(*
Implements the procedure for safely transitioning between device states by asserting the correct beam parameters for 
the state *)
FUNCTION_BLOCK BeamParameterTransitionManager
VAR_IN_OUT
	
	fbArbiter	:	FB_Arbiter;
	
END_VAR
VAR_INPUT
	i_TransitionAssertionID	:	UDINT := 0;
	i_stTransitionAssertion : ST_BeamParams := PMPS_GVL_BeamParams.cstSafeBeam; //Assertion required during transition (always safer than anything inbetween)
	
	i_nRequestedAssertionID	:	UDINT := 0;
	i_stRequestedAssertion	:	ST_BeamParams := PMPS_GVL_BeamParams.cstSafeBeam; //Requested assertion, change whenever
	
	i_xMoving	:	BOOL := FALSE; //Provide rising edge when device begins moving
	i_xDoneMoving	:	BOOL := FALSE; //Provide rising edge when device is done with a move
	
END_VAR
VAR_OUTPUT

	q_xTransitionAuthorized	:	BOOL := FALSE; //Rising edge indicating the device is safe to move, use as input to move execute (which requires a rising edge)

END_VAR

VAR
	nTargetAssertionID	:	UDINT := 0;
	stTargetAssertion	:	ST_BeamParams; //Current target assertion
	nCurrentAssertionID	:	UDINT := 0;
	
	xNewBP	:	BOOL;
	xTranBP	:	BOOL;
	xFinalBP	:	BOOL;
	
END_VAR

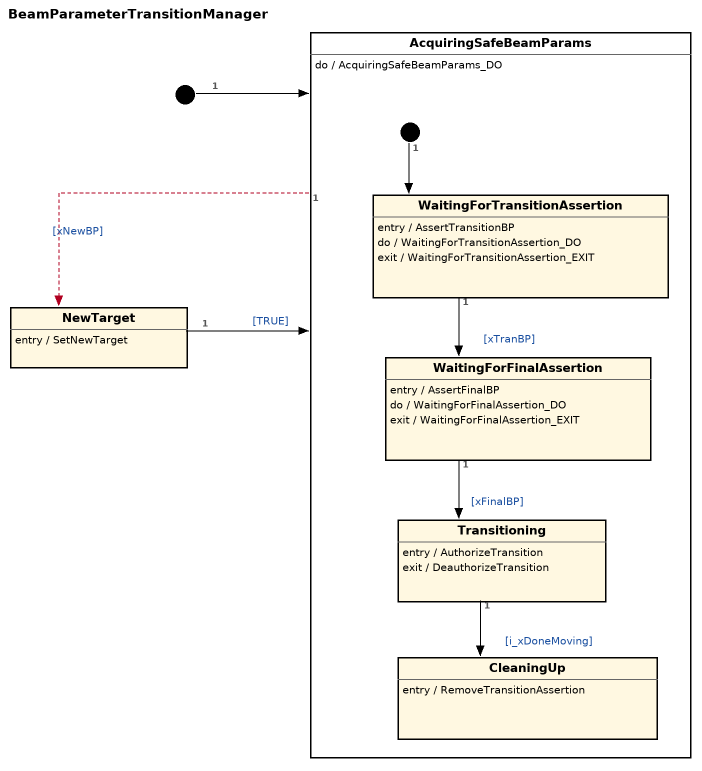
STATECHART BeamParameterTransitionManager  // abortable
    START StartState1_copy
    COMPOSITE STATE AcquiringSafeBeamParams
        do / AcquiringSafeBeamParams_DO
        START StartState1
        STATE WaitingForTransitionAssertion
            entry / AssertTransitionBP
            do / WaitingForTransitionAssertion_DO
            exit / WaitingForTransitionAssertion_EXIT
        STATE WaitingForFinalAssertion
            entry / AssertFinalBP
            do / WaitingForFinalAssertion_DO
            exit / WaitingForFinalAssertion_EXIT
        STATE Transitioning
            entry / AuthorizeTransition
            exit / DeauthorizeTransition
        STATE CleaningUp
            entry / RemoveTransitionAssertion
        StartState1 -> WaitingForTransitionAssertion  // priority 1, on completion
        WaitingForTransitionAssertion -> WaitingForFinalAssertion [xTranBP] // priority 1, rising edge
        WaitingForFinalAssertion -> Transitioning [xFinalBP] // priority 1, rising edge
        Transitioning -> CleaningUp [i_xDoneMoving] // priority 1, rising edge
    END_STATE
    STATE NewTarget
        entry / SetNewTarget
    StartState1_copy -> AcquiringSafeBeamParams  // priority 1, on completion
    AcquiringSafeBeamParams -> NewTarget [xNewBP] // priority 1, exception, rising edge
    NewTarget -> AcquiringSafeBeamParams [TRUE] // priority 1
END_STATECHART

ACTION AcquiringSafeBeamParams_DO:
xNewBP := nTargetAssertionID <> i_nRequestedAssertionID;
END_ACTION

ACTION AssertFinalBP:
//q_stFinalAssertion := stTargetAssertion;

//Clearing previous target parameters
(* This is considered safe at this step as the transition
state beam parameters should always be safer than the
current or target state beam parameters
*)
fbArbiter.A_RemoveAssertion( i_nStateID := nCurrentAssertionID );

//Asserting target parameters
fbArbiter.A_AssertBP(
	i_nStateID := nTargetAssertionID,
	i_stAssertBeamParams := stTargetAssertion
);

//Remembering final assertionID for removal later
nCurrentAssertionID := nTargetAssertionID;
END_ACTION

ACTION AssertTransitionBP:

fbArbiter.A_AssertBP(
	i_nStateID := i_TransitionAssertionID,
	i_stAssertBeamParams := i_stTransitionAssertion
);
END_ACTION

ACTION AuthorizeTransition:
q_xTransitionAuthorized := TRUE;
END_ACTION

ACTION DeauthorizeMove:

END_ACTION

ACTION DeauthorizeTransition:
q_xTransitionAuthorized := FALSE;
END_ACTION

ACTION RemoveTransitionAssertion:
//q_stTransitionAssertion := PMPS_GVL_BeamParams.cstFullBeam;

//Removing transition assertion
fbArbiter.A_RemoveAssertion( i_nStateID := i_TransitionAssertionID);



//TODO add something to verify removal
END_ACTION

ACTION RemoveTransitionAuthorization:

END_ACTION

ACTION SetNewTarget:
xNewBP := FALSE;
stTargetAssertion := i_stRequestedAssertion;
nTargetAssertionID := i_nRequestedAssertionID;
END_ACTION

ACTION WaitingForFinalAssertion_DO:
//Final Assertion Verification
fbArbiter.A_VerifyAssertion( i_nStateID := i_nRequestedAssertionID);
xFinalBP := F_SafeBPCompare(PMPS_GVL_BeamParams.stCurrentBeamParameters, stTargetAssertion) AND
	fbArbiter.q_xStateIDFound;
END_ACTION

ACTION WaitingForFinalAssertion_EXIT:
//Set this bool false so we can get a rising edge on the next try
xFinalBP := FALSE;
END_ACTION

ACTION WaitingForTransitionAssertion_DO:
//Transition Assertion Verification
fbArbiter.A_VerifyAssertion( i_nStateID := i_TransitionAssertionID); //TODO this may be an expensive operation as it's constantly checking the hashtable, could move it to be checked only when waitingfortransitionassertion
xTranBP	:= F_SafeBPCompare(PMPS_GVL_BeamParams.stCurrentBeamParameters, i_stTransitionAssertion) AND
	fbArbiter.q_xStateIDFound;
END_ACTION

ACTION WaitingForTransitionAssertion_EXIT:
xTranBP := FALSE;
END_ACTION

END_FUNCTION_BLOCK

(* stored: Version 1.1.0.1, ProductVersion 3.1.4022.12
   POU BeamParameterTransitionManager: Id {843312b6-3630-0fa6-1e20-da1ce4aaad4c}, SpecialFunc None
   Action AcquiringSafeBeamParams_DO: Id {603c4e25-97d2-01fd-3380-8f019adaa760}
   Action AssertFinalBP: Id {3aacecc4-95cc-0b9d-1f9c-d6c9dec8e836}
   Action AssertTransitionBP: Id {09eb738b-7411-0821-2e23-c9281e93e49d}
   Action AuthorizeTransition: Id {b727a18e-e395-0e7a-074b-b778698df218}
   Action DeauthorizeMove: Id {3b9e719b-fa51-0c03-3729-27bd539c56ba}
   Action DeauthorizeTransition: Id {85553ff9-652b-0f0d-38e0-23e9eece0909}
   Action RemoveTransitionAssertion: Id {fd3da30e-395a-0698-0f23-a3f0bc8df59f}
   Action RemoveTransitionAuthorization: Id {ad498ce1-478c-0d24-0076-296638013077}
   Action SetNewTarget: Id {cb54fd73-aaf3-0c05-2881-782da729c59b}
   Action WaitingForFinalAssertion_DO: Id {321877ce-1716-0d60-0edb-45fda6425ee5}
   Action WaitingForFinalAssertion_EXIT: Id {841774c7-aa1a-0f81-0d11-1d67419288e5}
   Action WaitingForTransitionAssertion_DO: Id {b28d9b59-2c93-0121-2340-e3e699a9fa4a}
   Action WaitingForTransitionAssertion_EXIT: Id {07d13c2b-9514-064a-3d0d-409feea20c70} *)
